// ---- POUs/PRG_IM1L1_PPM.TcPOU
PROGRAM PRG_IM1L1_PPM
VAR
    {attribute 'pytmc' := '
        pv: IM1L1:PPM
        io: io
    '}
    {attribute 'TcLinkTo' := '.fbGige.iIlluminatorINT := TIIB[IM1L1-EL4004]^AO Outputs Channel 1^Analog output;
                              .fbGige.bGigePower := TIIB[IM1L1-EL2004]^Channel 2^Output;
                              .fbPowerMeter.iVoltageINT := TIIB[IM1L1-EL3062]^AI Standard Channel 1^Value;
                              .fbPowerMeter.fbTempSensor.bError := TIIB[IM1L1-EL3314]^TC Inputs Channel 1^Status^Error;
                              .fbPowerMeter.fbTempSensor.bUnderrange := TIIB[IM1L1-EL3314]^TC Inputs Channel 1^Status^Underrange;
                              .fbPowerMeter.fbTempSensor.bOverrange := TIIB[IM1L1-EL3314]^TC Inputs Channel 1^Status^Overrange;
                              .fbPowerMeter.fbTempSensor.iRaw := TIIB[IM1L1-EL3314]^TC Inputs Channel 1^Value;
                              .fbYagTempSensor.bError := TIIB[IM1L1-EL3314]^TC Inputs Channel 2^Status^Error;
                              .fbYagTempSensor.bUnderrange := TIIB[IM1L1-EL3314]^TC Inputs Channel 2^Status^Underrange;
                              .fbYagTempSensor.bOverrange := TIIB[IM1L1-EL3314]^TC Inputs Channel 2^Status^Overrange;
                              .fbYagTempSensor.iRaw := TIIB[IM1L1-EL3314]^TC Inputs Channel 2^Value'}
    fbIM1L1: FB_PPM;

    fbStateSetup: FB_StateSetupHelper;
    stDefault: ST_PositionState := (
        fVelocity := 10,
        bMoveOk := TRUE,
        bValid := TRUE
    );
END_VAR


fbStateSetup(stPositionState:=stDefault, bSetDefault:=TRUE);
fbStateSetup(stPositionState:=fbIM1L1.stOut, fPosition:=-11,    sPmpsState:='IM1L1:PPM-OUT');
fbStateSetup(stPositionState:=fbIM1L1.stPower, fPosition:=-47.59, sPmpsState:='IM1L1:PPM-POWERMETER');
fbStateSetup(stPositionState:=fbIM1L1.stYag1, fPosition:=-71.69,  sPmpsState:='IM1L1:PPM-YAG1');
fbStateSetup(stPositionState:=fbIM1L1.stYag2, fPosition:=-97.70,  sPmpsState:='IM1L1:PPM-YAG2');

fbIM1L1(
    fbArbiter := GVL.fbArbiter2,
    fbFFHWO := GVL.fbFastFaultOutput2,
    stYStage := Main.M23,
    sDeviceName := 'IM1L1:PPM',
    sTransitionKey := 'IM1L1:PPM-TRANSITION',
    bEnableMotion := TRUE,
    bEnableBeamParams := TRUE,
    bEnablePositionLimits := TRUE,
    fResponsivity := 0.0640, //probably wrong, check with Phil
);

END_PROGRAM

// ---- POUs/PRG_IM2L0_XTES.TcPOU
PROGRAM PRG_IM2L0_XTES
VAR
    {attribute 'pytmc' := '
        pv: IM2L0:XTES
        io: io
    '}
    {attribute 'TcLinkTo' := '.bZoomEndFwd := TIIB[IM2L0-EL1088]^Channel 1^Input;
                              .bZoomEndBwd := TIIB[IM2L0-EL1088]^Channel 2^Input;
                              .bFocusEndFwd := TIIB[IM2L0-EL1088]^Channel 3^Input;
                              .bFocusEndBwd := TIIB[IM2L0-EL1088]^Channel 4^Input;
                              .fbOpal.bOpalPower := TIIB[IM2L0-EL2004]^Channel 2^Output;
                              .fbLED.bLedPower := TIIB[IM2L0-EL2004]^Channel 3^Output'}
    fbIM2L0: FB_XPIM;
    {attribute 'TcLinkTo' := '.Status := TIIB[IM2L0-EL6002]^COM TxPDO-Map Inputs Channel 1^Status;
                              .D[0] := TIIB[IM2L0-EL6002]^COM TxPDO-Map Inputs Channel 1^Data In 0;
                              .D[1] := TIIB[IM2L0-EL6002]^COM TxPDO-Map Inputs Channel 1^Data In 1;
                              .D[2] := TIIB[IM2L0-EL6002]^COM TxPDO-Map Inputs Channel 1^Data In 2;
                              .D[3] := TIIB[IM2L0-EL6002]^COM TxPDO-Map Inputs Channel 1^Data In 3;
                              .D[4] := TIIB[IM2L0-EL6002]^COM TxPDO-Map Inputs Channel 1^Data In 4;
                              .D[5] := TIIB[IM2L0-EL6002]^COM TxPDO-Map Inputs Channel 1^Data In 5;
                              .D[6] := TIIB[IM2L0-EL6002]^COM TxPDO-Map Inputs Channel 1^Data In 6;
                              .D[7] := TIIB[IM2L0-EL6002]^COM TxPDO-Map Inputs Channel 1^Data In 7;
                              .D[8] := TIIB[IM2L0-EL6002]^COM TxPDO-Map Inputs Channel 1^Data In 8;
                              .D[9] := TIIB[IM2L0-EL6002]^COM TxPDO-Map Inputs Channel 1^Data In 9;
                              .D[10] := TIIB[IM2L0-EL6002]^COM TxPDO-Map Inputs Channel 1^Data In 10;
                              .D[11] := TIIB[IM2L0-EL6002]^COM TxPDO-Map Inputs Channel 1^Data In 11;
                              .D[12] := TIIB[IM2L0-EL6002]^COM TxPDO-Map Inputs Channel 1^Data In 12;
                              .D[13] := TIIB[IM2L0-EL6002]^COM TxPDO-Map Inputs Channel 1^Data In 13;
                              .D[14] := TIIB[IM2L0-EL6002]^COM TxPDO-Map Inputs Channel 1^Data In 14;
                              .D[15] := TIIB[IM2L0-EL6002]^COM TxPDO-Map Inputs Channel 1^Data In 15;
                              .D[16] := TIIB[IM2L0-EL6002]^COM TxPDO-Map Inputs Channel 1^Data In 16;
                              .D[17] := TIIB[IM2L0-EL6002]^COM TxPDO-Map Inputs Channel 1^Data In 17;
                              .D[18] := TIIB[IM2L0-EL6002]^COM TxPDO-Map Inputs Channel 1^Data In 18;
                              .D[19] := TIIB[IM2L0-EL6002]^COM TxPDO-Map Inputs Channel 1^Data In 19;
                              .D[20] := TIIB[IM2L0-EL6002]^COM TxPDO-Map Inputs Channel 1^Data In 20;
                              .D[21] := TIIB[IM2L0-EL6002]^COM TxPDO-Map Inputs Channel 1^Data In 21'}
    stEL6In AT %I*: EL6InData22b;
    {attribute 'TcLinkTo' := '.Ctrl := TIIB[IM2L0-EL6002]^COM RxPDO-Map Outputs Channel 1^Ctrl;
                              .D[0] := TIIB[IM2L0-EL6002]^COM RxPDO-Map Outputs Channel 1^Data Out 0;
                              .D[1] := TIIB[IM2L0-EL6002]^COM RxPDO-Map Outputs Channel 1^Data Out 1;
                              .D[2] := TIIB[IM2L0-EL6002]^COM RxPDO-Map Outputs Channel 1^Data Out 2;
                              .D[3] := TIIB[IM2L0-EL6002]^COM RxPDO-Map Outputs Channel 1^Data Out 3;
                              .D[4] := TIIB[IM2L0-EL6002]^COM RxPDO-Map Outputs Channel 1^Data Out 4;
                              .D[5] := TIIB[IM2L0-EL6002]^COM RxPDO-Map Outputs Channel 1^Data Out 5;
                              .D[6] := TIIB[IM2L0-EL6002]^COM RxPDO-Map Outputs Channel 1^Data Out 6;
                              .D[7] := TIIB[IM2L0-EL6002]^COM RxPDO-Map Outputs Channel 1^Data Out 7;
                              .D[8] := TIIB[IM2L0-EL6002]^COM RxPDO-Map Outputs Channel 1^Data Out 8;
                              .D[9] := TIIB[IM2L0-EL6002]^COM RxPDO-Map Outputs Channel 1^Data Out 9;
                              .D[10] := TIIB[IM2L0-EL6002]^COM RxPDO-Map Outputs Channel 1^Data Out 10;
                              .D[11] := TIIB[IM2L0-EL6002]^COM RxPDO-Map Outputs Channel 1^Data Out 11;
                              .D[12] := TIIB[IM2L0-EL6002]^COM RxPDO-Map Outputs Channel 1^Data Out 12;
                              .D[13] := TIIB[IM2L0-EL6002]^COM RxPDO-Map Outputs Channel 1^Data Out 13;
                              .D[14] := TIIB[IM2L0-EL6002]^COM RxPDO-Map Outputs Channel 1^Data Out 14;
                              .D[15] := TIIB[IM2L0-EL6002]^COM RxPDO-Map Outputs Channel 1^Data Out 15;
                              .D[16] := TIIB[IM2L0-EL6002]^COM RxPDO-Map Outputs Channel 1^Data Out 16;
                              .D[17] := TIIB[IM2L0-EL6002]^COM RxPDO-Map Outputs Channel 1^Data Out 17;
                              .D[18] := TIIB[IM2L0-EL6002]^COM RxPDO-Map Outputs Channel 1^Data Out 18;
                              .D[19] := TIIB[IM2L0-EL6002]^COM RxPDO-Map Outputs Channel 1^Data Out 19;
                              .D[20] := TIIB[IM2L0-EL6002]^COM RxPDO-Map Outputs Channel 1^Data Out 20;
                              .D[21] := TIIB[IM2L0-EL6002]^COM RxPDO-Map Outputs Channel 1^Data Out 21'}
    stEL6Out AT %Q*: EL6OutData22b;

    fbStateSetup: FB_StateSetupHelper;
    stDefault: ST_PositionState := (
        fVelocity := 1,
        bMoveOk := TRUE,
        bValid := TRUE
    );

    {attribute 'TcLinkTo' := 'TIIB[IM2L0-EL7041]^STM Status^Status^Digital input 1'}
    bDefectiveLimitSwitch AT %I*: BOOL;
END_VAR


fbStateSetup(stPositionState:=stDefault, bSetDefault:=TRUE);
fbStateSetup(stPositionState:=fbIM2L0.stOut, fPosition:=0,          sPmpsState:='IM2L0:XTES-OUT');
fbStateSetup(stPositionState:=fbIM2L0.stYag, fPosition:=-87.65,     sPmpsState:='IM2L0:XTES-YAG');
fbStateSetup(stPositionState:=fbIM2L0.stDiamond, fPosition:=-57.65, sPmpsState:='IM2L0:XTES-DIAMOND');
fbStateSetup(stPositionState:=fbIM2L0.stReticle, fPosition:=-27.65, sPmpsState:='IM2L0:XTES-RETICLE');

Main.M24.bLimitForwardEnable := bDefectiveLimitSwitch OR (Main.M24.stAxisStatus.fActPosition < 0);

fbIM2L0(
    fbArbiter := GVL.fbArbiter,
    fbFFHWO := GVL.fbFastFaultOutput1,
    stYStage := Main.M24,
    stZoomStage := Main.M25,
    stFocusStage := Main.M26,
    stEl6In := stEL6In,
    stEl6Out := stEl6Out,
    sDeviceName := 'IM2L0:XTES',
    sTransitionKey := 'IM2L0:XTES-TRANSITION',
    bEnableMotion := TRUE,
    bEnableBeamParams := TRUE,
    bEnablePositionLimits := TRUE,
);

END_PROGRAM

// ---- POUs/PRG_IM3L0_PPM.TcPOU
PROGRAM PRG_IM3L0_PPM
VAR
    {attribute 'pytmc' := '
        pv: IM3L0:PPM
        io: io
    '}
    {attribute 'TcLinkTo' := '.fbGige.iIlluminatorINT := TIIB[IM3L0-EL4004]^AO Outputs Channel 1^Analog output;
                              .fbGige.bGigePower := TIIB[IM3L0-EL2004]^Channel 2^Output;
                              .fbPowerMeter.iVoltageINT := TIIB[IM3L0-EL3062]^AI Standard Channel 1^Value;
                              .fbPowerMeter.fbTempSensor.bError := TIIB[IM3L0-EL3314]^TC Inputs Channel 1^Status^Error;
                              .fbPowerMeter.fbTempSensor.bUnderrange := TIIB[IM3L0-EL3314]^TC Inputs Channel 1^Status^Underrange;
                              .fbPowerMeter.fbTempSensor.bOverrange := TIIB[IM3L0-EL3314]^TC Inputs Channel 1^Status^Overrange;
                              .fbPowerMeter.fbTempSensor.iRaw := TIIB[IM3L0-EL3314]^TC Inputs Channel 1^Value;
                              .fbYagTempSensor.bError := TIIB[IM3L0-EL3314]^TC Inputs Channel 2^Status^Error;
                              .fbYagTempSensor.bUnderrange := TIIB[IM3L0-EL3314]^TC Inputs Channel 2^Status^Underrange;
                              .fbYagTempSensor.bOverrange := TIIB[IM3L0-EL3314]^TC Inputs Channel 2^Status^Overrange;
                              .fbYagTempSensor.iRaw := TIIB[IM3L0-EL3314]^TC Inputs Channel 2^Value'}
    fbIM3L0: FB_PPM;

    fbStateSetup: FB_StateSetupHelper;
    stDefault: ST_PositionState := (
        fVelocity := 10,
        bMoveOk := TRUE,
        bValid := TRUE
    );
END_VAR


fbStateSetup(stPositionState:=stDefault, bSetDefault:=TRUE);
fbStateSetup(stPositionState:=fbIM3L0.stOut, fPosition:=-8.40,    sPmpsState:='IM3L0:PPM-OUT');
fbStateSetup(stPositionState:=fbIM3L0.stPower, fPosition:=-47.40, sPmpsState:='IM3L0:PPM-POWERMETER');
fbStateSetup(stPositionState:=fbIM3L0.stYag1, fPosition:=-71.50,  sPmpsState:='IM3L0:PPM-YAG1');
fbStateSetup(stPositionState:=fbIM3L0.stYag2, fPosition:=-97.51,  sPmpsState:='IM3L0:PPM-YAG2');

fbIM3L0(
    fbArbiter := GVL.fbArbiter,
    fbFFHWO := GVL.fbFastFaultOutput1,
    stYStage := Main.M27,
    sDeviceName := 'IM3L0:PPM',
    sTransitionKey := 'IM3L0:PPM-TRANSITION',
    bEnableMotion := TRUE,
    bEnableBeamParams := TRUE,
    bEnablePositionLimits := TRUE,
    fResponsivity := 0.0506,
);

END_PROGRAM

// ---- POUs/PRG_IM4L0_XTES.TcPOU
PROGRAM PRG_IM4L0_XTES
VAR
    {attribute 'pytmc' := '
        pv: IM4L0:XTES
        io: io
    '}
    {attribute 'TcLinkTo' := '.bZoomEndFwd := TIIB[IM4L0-EL1088]^Channel 1^Input;
                              .bZoomEndBwd := TIIB[IM4L0-EL1088]^Channel 2^Input;
                              .bFocusEndFwd := TIIB[IM4L0-EL1088]^Channel 3^Input;
                              .bFocusEndBwd := TIIB[IM4L0-EL1088]^Channel 4^Input;
                              .fbOpal.bOpalPower := TIIB[IM4L0-EL2004]^Channel 2^Output;
                              .fbLED.bLedPower := TIIB[IM4L0-EL2004]^Channel 3^Output'}
    fbIM4L0: FB_XPIM;
    {attribute 'TcLinkTo' := '.Status := TIIB[IM4L0-EL6002]^COM TxPDO-Map Inputs Channel 1^Status;
                              .D[0] := TIIB[IM4L0-EL6002]^COM TxPDO-Map Inputs Channel 1^Data In 0;
                              .D[1] := TIIB[IM4L0-EL6002]^COM TxPDO-Map Inputs Channel 1^Data In 1;
                              .D[2] := TIIB[IM4L0-EL6002]^COM TxPDO-Map Inputs Channel 1^Data In 2;
                              .D[3] := TIIB[IM4L0-EL6002]^COM TxPDO-Map Inputs Channel 1^Data In 3;
                              .D[4] := TIIB[IM4L0-EL6002]^COM TxPDO-Map Inputs Channel 1^Data In 4;
                              .D[5] := TIIB[IM4L0-EL6002]^COM TxPDO-Map Inputs Channel 1^Data In 5;
                              .D[6] := TIIB[IM4L0-EL6002]^COM TxPDO-Map Inputs Channel 1^Data In 6;
                              .D[7] := TIIB[IM4L0-EL6002]^COM TxPDO-Map Inputs Channel 1^Data In 7;
                              .D[8] := TIIB[IM4L0-EL6002]^COM TxPDO-Map Inputs Channel 1^Data In 8;
                              .D[9] := TIIB[IM4L0-EL6002]^COM TxPDO-Map Inputs Channel 1^Data In 9;
                              .D[10] := TIIB[IM4L0-EL6002]^COM TxPDO-Map Inputs Channel 1^Data In 10;
                              .D[11] := TIIB[IM4L0-EL6002]^COM TxPDO-Map Inputs Channel 1^Data In 11;
                              .D[12] := TIIB[IM4L0-EL6002]^COM TxPDO-Map Inputs Channel 1^Data In 12;
                              .D[13] := TIIB[IM4L0-EL6002]^COM TxPDO-Map Inputs Channel 1^Data In 13;
                              .D[14] := TIIB[IM4L0-EL6002]^COM TxPDO-Map Inputs Channel 1^Data In 14;
                              .D[15] := TIIB[IM4L0-EL6002]^COM TxPDO-Map Inputs Channel 1^Data In 15;
                              .D[16] := TIIB[IM4L0-EL6002]^COM TxPDO-Map Inputs Channel 1^Data In 16;
                              .D[17] := TIIB[IM4L0-EL6002]^COM TxPDO-Map Inputs Channel 1^Data In 17;
                              .D[18] := TIIB[IM4L0-EL6002]^COM TxPDO-Map Inputs Channel 1^Data In 18;
                              .D[19] := TIIB[IM4L0-EL6002]^COM TxPDO-Map Inputs Channel 1^Data In 19;
                              .D[20] := TIIB[IM4L0-EL6002]^COM TxPDO-Map Inputs Channel 1^Data In 20;
                              .D[21] := TIIB[IM4L0-EL6002]^COM TxPDO-Map Inputs Channel 1^Data In 21'}
    stEL6In AT %I*: EL6InData22b;
    {attribute 'TcLinkTo' := '.Ctrl := TIIB[IM4L0-EL6002]^COM RxPDO-Map Outputs Channel 1^Ctrl;
                              .D[0] := TIIB[IM4L0-EL6002]^COM RxPDO-Map Outputs Channel 1^Data Out 0;
                              .D[1] := TIIB[IM4L0-EL6002]^COM RxPDO-Map Outputs Channel 1^Data Out 1;
                              .D[2] := TIIB[IM4L0-EL6002]^COM RxPDO-Map Outputs Channel 1^Data Out 2;
                              .D[3] := TIIB[IM4L0-EL6002]^COM RxPDO-Map Outputs Channel 1^Data Out 3;
                              .D[4] := TIIB[IM4L0-EL6002]^COM RxPDO-Map Outputs Channel 1^Data Out 4;
                              .D[5] := TIIB[IM4L0-EL6002]^COM RxPDO-Map Outputs Channel 1^Data Out 5;
                              .D[6] := TIIB[IM4L0-EL6002]^COM RxPDO-Map Outputs Channel 1^Data Out 6;
                              .D[7] := TIIB[IM4L0-EL6002]^COM RxPDO-Map Outputs Channel 1^Data Out 7;
                              .D[8] := TIIB[IM4L0-EL6002]^COM RxPDO-Map Outputs Channel 1^Data Out 8;
                              .D[9] := TIIB[IM4L0-EL6002]^COM RxPDO-Map Outputs Channel 1^Data Out 9;
                              .D[10] := TIIB[IM4L0-EL6002]^COM RxPDO-Map Outputs Channel 1^Data Out 10;
                              .D[11] := TIIB[IM4L0-EL6002]^COM RxPDO-Map Outputs Channel 1^Data Out 11;
                              .D[12] := TIIB[IM4L0-EL6002]^COM RxPDO-Map Outputs Channel 1^Data Out 12;
                              .D[13] := TIIB[IM4L0-EL6002]^COM RxPDO-Map Outputs Channel 1^Data Out 13;
                              .D[14] := TIIB[IM4L0-EL6002]^COM RxPDO-Map Outputs Channel 1^Data Out 14;
                              .D[15] := TIIB[IM4L0-EL6002]^COM RxPDO-Map Outputs Channel 1^Data Out 15;
                              .D[16] := TIIB[IM4L0-EL6002]^COM RxPDO-Map Outputs Channel 1^Data Out 16;
                              .D[17] := TIIB[IM4L0-EL6002]^COM RxPDO-Map Outputs Channel 1^Data Out 17;
                              .D[18] := TIIB[IM4L0-EL6002]^COM RxPDO-Map Outputs Channel 1^Data Out 18;
                              .D[19] := TIIB[IM4L0-EL6002]^COM RxPDO-Map Outputs Channel 1^Data Out 19;
                              .D[20] := TIIB[IM4L0-EL6002]^COM RxPDO-Map Outputs Channel 1^Data Out 20;
                              .D[21] := TIIB[IM4L0-EL6002]^COM RxPDO-Map Outputs Channel 1^Data Out 21'}
    stEL6Out AT %Q*: EL6OutData22b;

     {attribute 'pytmc' := 'pv: IM4L0:SCRP:LED:01:PWR
                        io: io
                        field: ZNAM OFF
                        field: ONAM ON
     '}

     {attribute 'TcLinkTo' := 'TIIB[IM4L0-EL2004]^Channel 4^Output'}
    bIM4L0_SCRP_LED_01 AT %Q*: BOOL;

    fbStateSetup: FB_StateSetupHelper;
    stDefault: ST_PositionState := (
        fVelocity := 1,
        bMoveOk := TRUE,
        bValid := TRUE
    );
END_VAR


fbStateSetup(stPositionState:=stDefault, bSetDefault:=TRUE);
fbStateSetup(stPositionState:=fbIM4L0.stOut, fPosition:=0,          sPmpsState:='IM4L0:XTES-OUT');
fbStateSetup(stPositionState:=fbIM4L0.stYag, fPosition:=-86.65,     sPmpsState:='IM4L0:XTES-YAG');
fbStateSetup(stPositionState:=fbIM4L0.stDiamond, fPosition:=-56.65, sPmpsState:='IM4L0:XTES-DIAMOND');
fbStateSetup(stPositionState:=fbIM4L0.stReticle, fPosition:=-26.65, sPmpsState:='IM4L0:XTES-RETICLE');

fbIM4L0(
    fbArbiter := GVL.fbArbiter,
    fbFFHWO := GVL.fbFastFaultOutput1,
    stYStage := Main.M28,
    stZoomStage := Main.M29,
    stFocusStage := Main.M30,
    stEl6In := stEL6In,
    stEl6Out := stEl6Out,
    sDeviceName := 'IM4L0:XTES',
    sTransitionKey := 'IM4L0:XTES-TRANSITION',
    bEnableMotion := TRUE,
    bEnableBeamParams := TRUE,
    bEnablePositionLimits := TRUE,
);

END_PROGRAM

// ---- POUs/PRG_PF1L0_WFS.TcPOU
PROGRAM PRG_PF1L0_WFS
VAR
    {attribute 'pytmc' := '
        pv: PF1L0:WFS
        io: io
    '}
    {attribute 'TcLinkTo' := '.fbThermoCouple1.bError := TIIB[PF1L0-EL3314]^TC Inputs Channel 1^Status^Error;
                              .fbThermoCouple1.bUnderrange := TIIB[PF1L0-EL3314]^TC Inputs Channel 1^Status^Underrange;
                              .fbThermoCouple1.bOverrange := TIIB[PF1L0-EL3314]^TC Inputs Channel 1^Status^Overrange;
                              .fbThermoCouple1.iRaw := TIIB[PF1L0-EL3314]^TC Inputs Channel 1^Value;
                              .fbThermoCouple2.bError := TIIB[PF1L0-EL3314]^TC Inputs Channel 2^Status^Error;
                              .fbThermoCouple2.bUnderrange := TIIB[PF1L0-EL3314]^TC Inputs Channel 2^Status^Underrange;
                              .fbThermoCouple2.bOverrange := TIIB[PF1L0-EL3314]^TC Inputs Channel 2^Status^Overrange;
                              .fbThermoCouple2.iRaw := TIIB[PF1L0-EL3314]^TC Inputs Channel 2^Value'}
    fbPF1L0: FB_WFS;
    stSiBP: ST_BeamParams := PMPS_GVL.cstFullBeam;
    stFoilBP: ST_BeamParams := PMPS_GVL.cstFullBeam;

    fbStateSetup: FB_StateSetupHelper;
    stDefault: ST_PositionState := (
        fVelocity := 1,
        bMoveOk := TRUE,
        bValid := TRUE
    );
END_VAR


fbStateSetup(stPositionState:=stDefault, bSetDefault:=TRUE);
fbStateSetup(stPositionState:=fbPF1L0.stOut, fPosition:=-13,         sPmpsState:='PF1L0:WFS-OUT');
fbStateSetup(stPositionState:=fbPF1L0.stTarget1, fPosition:=-93.77,  sPmpsState:='PF1L0:WFS-TARGET1');
fbStateSetup(stPositionState:=fbPF1L0.stTarget2, fPosition:=-79.402, sPmpsState:='PF1L0:WFS-TARGET2');
fbStateSetup(stPositionState:=fbPF1L0.stTarget3, fPosition:=-65.028, sPmpsState:='PF1L0:WFS-TARGET3');
fbStateSetup(stPositionState:=fbPF1L0.stTarget4, fPosition:=-50.652, sPmpsState:='PF1L0:WFS-TARGET4');
fbStateSetup(stPositionState:=fbPF1L0.stTarget5, fPosition:=-36.277, sPmpsState:='PF1L0:WFS-TARGET5');

fbPF1L0(
    fbArbiter := GVL.fbArbiter,
    fbFFHWO := GVL.fbFastFaultOutput1,
    stYStage := Main.M31,
    stZStage := Main.M32,
    sDeviceName := 'PF1L0:WFS',
    sTransitionKey := 'PF1L0:WFS-TRANSITION',
    bEnableMotion := TRUE,
    bEnableBeamParams := TRUE,
    bEnablePositionLimits := TRUE,
    eEnumGet => GVL.ePF1L0State,
);

END_PROGRAM

// ---- POUs/PRG_RTDSL0.TcPOU
PROGRAM PRG_RTDSL0
VAR

    fbRTDSL0_Diode_MMS_01: FB_MotionStage;

    bInit: BOOL := TRUE;
END_VAR

// Placeholder, standard simulated motion for all axes
//fbMotion1(stMotionStage := Main.M33);
//fbMotion2(stMotionStage := Main.M34);
//fbMotion3(stMotionStage := Main.M35);
//fbMotion4(stMotionStage := Main.M36);
//fbMotion5(stMotionStage := Main.M37);
//fbMotion6(stMotionStage := Main.M38);
//fbMotion7(stMotionStage := Main.M39);

//Pneumatic actuators - OTR filters

RTDSL0_MPA_01(
    ibInsertOK:= TRUE,
    ibRetractOK:= TRUE ,
    ibPMPS_OK:= TRUE ,
    ibOverrideInterlock:= ,
    q_stAct=> ,
    xMPS_OK=> ,
    xDone=> ,
    i_xReset := ,
    io_fbFFHWO := GVL.fbFastFaultOutput1,
    bEnableFF := TRUE,
);

RTDSL0_MPA_02(
    ibInsertOK:= TRUE,
    ibRetractOK:= TRUE ,
    ibPMPS_OK:= TRUE ,
    ibOverrideInterlock:= ,
    q_stAct=> ,
    xMPS_OK=> ,
    xDone=> ,
    i_xReset := ,
    io_fbFFHWO := GVL.fbFastFaultOutput1,
    bEnableFF := TRUE,
);

RTDSL0_MPA_03(
    ibInsertOK:= TRUE,
    ibRetractOK:= TRUE ,
    ibPMPS_OK:= TRUE ,
    ibOverrideInterlock:= ,
    q_stAct=> ,
    xMPS_OK=> ,
    xDone=> ,
    i_xReset := ,
    io_fbFFHWO := GVL.fbFastFaultOutput1,
    bEnableFF := FALSE,
);
//  init the motion stages parameters
IF ( bInit) THEN
    Main.M33.bHardwareEnable := TRUE;
    Main.M33.bPowerSelf :=TRUE;
    Main.M33.nBrakeMode := ENUM_StageBrakeMode.NO_BRAKE;
    (* uncomment when mccallister goes from RTDSK0 -> RTDSL0
    Main.M34.bHardwareEnable := TRUE;
    Main.M34.bPowerSelf :=TRUE;
    Main.M34.nBrakeMode := ENUM_StageBrakeMode.NO_BRAKE;

    Main.M35.bHardwareEnable := TRUE;
    Main.M35.bPowerSelf :=TRUE;
    Main.M35.nBrakeMode := ENUM_StageBrakeMode.NO_BRAKE;

    Main.M36.bHardwareEnable := TRUE;
    Main.M36.bPowerSelf :=TRUE;
    Main.M36.nBrakeMode := ENUM_StageBrakeMode.NO_BRAKE;

    //LDM motor
    Main.M37.bHardwareEnable := TRUE;
    Main.M37.bPowerSelf :=TRUE;
    Main.M37.nBrakeMode := ENUM_StageBrakeMode.NO_BRAKE;
    *)
    Main.M33.nHomingMode := ENUM_EpicsHomeCmd.HIGH_LIMIT;
    //uncomment when mccallister gets moved RTDSK0->RTDSL0
    //Main.M34.nHomingMode := ENUM_EpicsHomeCmd.HIGH_LIMIT;
    //Main.M35.nHomingMode := ENUM_EpicsHomeCmd.HIGH_LIMIT;
    //Main.M36.nHomingMode := ENUM_EpicsHomeCmd.HIGH_LIMIT;
    Main.M37.nHomingMode := ENUM_EpicsHomeCmd.HIGH_LIMIT;

        bInit := FALSE;

END_IF


fbRTDSL0_Diode_MMS_01 (stMotionStage := Main.M33);
//uncomment when mccallister stage RTDSK0 -> RTDSL0
//fbRTDSL0_SCRP_MMS_01 (stMotionStage := Main.M34);
//fbRTDSL0_SCRP_MMS_02 (stMotionStage := Main.M35);
//fbRTDSL0_SCRP_MMS_03 (stMotionStage := Main.M36);
//fbRTDSL0_LDM_MMS_01 (stMotionStage := Main.M37);
//uncomment when mccallister stage RTDSK0->RTDSL0
//fbRTDSK0_SCRP_LED_01 (enumXPIM := Main.LED1);

END_PROGRAM

// ---- POUs/PRG_SL1L0_POWER.TcPOU
PROGRAM PRG_SL1L0_POWER
VAR // fix linking to rtd in the following order Bottom - South - TOP - NORTH
    {attribute 'pytmc' := '
        pv: SL1L0:POWER
        io: io
    '}
    {attribute 'TcLinkTo' := '.RTD_Bottom_1.iRaw := TIIB[SL1L0-EL3202-E8]^RTD Inputs Channel 1^Value;
                              .RTD_Bottom_1.bError := TIIB[SL1L0-EL3202-E8]^RTD Inputs Channel 1^Status^Error;
                              .RTD_Bottom_1.bUnderrange := TIIB[SL1L0-EL3202-E8]^RTD Inputs Channel 1^Status^Underrange;
                              .RTD_Bottom_1.bOverrange := TIIB[SL1L0-EL3202-E8]^RTD Inputs Channel 1^Status^Overrange;
                              .RTD_Bottom_2.iRaw := TIIB[SL1L0-EL3202-E8]^RTD Inputs Channel 2^Value;
                              .RTD_Bottom_2.bError := TIIB[SL1L0-EL3202-E8]^RTD Inputs Channel 2^Status^Error;
                              .RTD_Bottom_2.bUnderrange := TIIB[SL1L0-EL3202-E8]^RTD Inputs Channel 2^Status^Underrange;
                              .RTD_Bottom_2.bOverrange := TIIB[SL1L0-EL3202-E8]^RTD Inputs Channel 2^Status^Overrange;
                              .RTD_South_1.iRaw := TIIB[SL1L0-EL3202-E9]^RTD Inputs Channel 1^Value;
                              .RTD_South_1.bError := TIIB[SL1L0-EL3202-E9]^RTD Inputs Channel 1^Status^Error;
                              .RTD_South_1.bUnderrange := TIIB[SL1L0-EL3202-E9]^RTD Inputs Channel 1^Status^Underrange;
                              .RTD_South_1.bOverrange := TIIB[SL1L0-EL3202-E9]^RTD Inputs Channel 1^Status^Overrange;
                              .RTD_South_2.iRaw := TIIB[SL1L0-EL3202-E9]^RTD Inputs Channel 2^Value;
                              .RTD_South_2.bError := TIIB[SL1L0-EL3202-E9]^RTD Inputs Channel 2^Status^Error;
                              .RTD_South_2.bUnderrange := TIIB[SL1L0-EL3202-E9]^RTD Inputs Channel 2^Status^Underrange;
                              .RTD_South_2.bOverrange := TIIB[SL1L0-EL3202-E9]^RTD Inputs Channel 2^Status^Overrange;
                              .RTD_TOP_1.iRaw := TIIB[SL1L0-EL3202-E10]^RTD Inputs Channel 1^Value;
                              .RTD_TOP_1.bError := TIIB[SL1L0-EL3202-E10]^RTD Inputs Channel 1^Status^Error;
                              .RTD_TOP_1.bUnderrange := TIIB[SL1L0-EL3202-E10]^RTD Inputs Channel 1^Status^Underrange;
                              .RTD_TOP_1.bOverrange := TIIB[SL1L0-EL3202-E10]^RTD Inputs Channel 1^Status^Overrange;
                              .RTD_TOP_2.iRaw := TIIB[SL1L0-EL3202-E10]^RTD Inputs Channel 2^Value;
                              .RTD_TOP_2.bError := TIIB[SL1L0-EL3202-E10]^RTD Inputs Channel 2^Status^Error;
                              .RTD_TOP_2.bUnderrange := TIIB[SL1L0-EL3202-E10]^RTD Inputs Channel 2^Status^Underrange;
                              .RTD_TOP_2.bOverrange := TIIB[SL1L0-EL3202-E10]^RTD Inputs Channel 2^Status^Overrange;
                              .RTD_North_1.iRaw := TIIB[SL1L0-EL3202-E11]^RTD Inputs Channel 1^Value;
                              .RTD_North_1.bError := TIIB[SL1L0-EL3202-E11]^RTD Inputs Channel 1^Status^Error;
                              .RTD_North_1.bUnderrange := TIIB[SL1L0-EL3202-E11]^RTD Inputs Channel 1^Status^Underrange;
                              .RTD_North_1.bOverrange := TIIB[SL1L0-EL3202-E11]^RTD Inputs Channel 1^Status^Overrange;
                              .RTD_North_2.iRaw := TIIB[SL1L0-EL3202-E11]^RTD Inputs Channel 2^Value;
                              .RTD_North_2.bError := TIIB[SL1L0-EL3202-E11]^RTD Inputs Channel 2^Status^Error;
                              .RTD_North_2.bUnderrange := TIIB[SL1L0-EL3202-E11]^RTD Inputs Channel 2^Status^Underrange;
                              .RTD_North_2.bOverrange := TIIB[SL1L0-EL3202-E11]^RTD Inputs Channel 2^Status^Overrange'}
    fbSL1L0: FB_SLITS_POWER;

    {attribute 'pytmc' := '
    pv: SL1L0:POWER:GO;
    io: io;
    field: ZNAM False;
    field: ONAM True;
    '}
    bExecuteMotion:BOOL ;

    // Default True until it is properly linked to PMPS bit
    bMoveOk:BOOL :=TRUE;


    mcPower : ARRAY [1..4] OF MC_POWER;

        (*Offsets*)
    (* Absolute encoder value at the HLS + Absolute encoder value at the centered beam *)
    rEncoderOffsetTop: REAL := 15.55;
    rEncoderOffsetBottom: REAL := -12.99;
    rEncoderOffsetNorth: REAL := 12.2;
    rEncoderOffsetSouth: REAL := -16.8;

END_VAR



(*
--MAPPING TO PHYSICAL TERMINAL--
Main.41 -> M1    (Bottom)
Main.42 -> M2    (South)
Main.43 -> M3    (Top)
Main.44 -> M4    (North)
*)

fbSL1L0.rEncoderOffsetTop := rEncoderOffsetTop;
fbSL1L0.rEncoderOffsetBottom := rEncoderOffsetBottom;
fbSL1L0.rEncoderOffsetNorth := rEncoderOffsetNorth;
fbSL1L0.rEncoderOffsetSouth := rEncoderOffsetSouth;

//fbSL1L0.bExecuteMotion := bExecuteMotion;
fbSL1L0.bMoveOk := bMoveOk;
fbSL1L0(stTopBlade:=  Main.M43,
        stBottomBlade:= Main.M41,
        stNorthBlade:=  Main.M44,
        stSouthBlade:=  Main.M42,
        bExecuteMotion:=bExecuteMotion,
        io_fbFFHWO := GVL.fbFastFaultOutput1,
        fbArbiter := GVL.fbArbiter,
);
//fbSL1L0.M_UpdatePMPS(1); Not sure what index to use

//for testing purposes only. comment-out/delete once done.
(*mcPower[1](axis:=Main.M41.Axis, Enable:=TRUE, enable_positive:=Main.M41.bLimitForwardEnable, enable_negative:=Main.M41.bLimitBackwardEnable);
mcPower[2](axis:=Main.M42.Axis, Enable:=TRUE, enable_positive:=Main.M42.bLimitForwardEnable, enable_negative:=Main.M42.bLimitBackwardEnable);
mcPower[3](axis:=Main.M43.Axis, Enable:=TRUE, enable_positive:=Main.M43.bLimitForwardEnable, enable_negative:=Main.M43.bLimitBackwardEnable);
mcPower[4](axis:=Main.M44.Axis, Enable:=TRUE, enable_positive:=Main.M44.bLimitForwardEnable, enable_negative:=Main.M44.bLimitBackwardEnable);*)

END_PROGRAM

// ---- Temp/FB_SLITS_POWER.TcPOU
FUNCTION_BLOCK FB_SLITS_POWER EXTENDS FB_SLITS
VAR_INPUT
END_VAR
VAR
     {attribute 'pytmc' := '
        pv: FSW
    '}
    fbFlowSwitch: FB_XTES_Flowswitch;


    //RTDs
    {attribute 'pytmc' := '
        pv: TOP:RTD:01
    '}
    RTD_TOP_1: FB_TempSensor;
    {attribute 'pytmc' := '
        pv: TOP:RTD:02
    '}
    RTD_TOP_2: FB_TempSensor;
    {attribute 'pytmc' := '
        pv: BOTTOM:RTD:01
    '}
    RTD_Bottom_1: FB_TempSensor;
    {attribute 'pytmc' := '
        pv: BOTTOM:RTD:02
    '}
    RTD_Bottom_2: FB_TempSensor;

    {attribute 'pytmc' := '
        pv: NORTH:RTD:01
    '}
    RTD_North_1: FB_TempSensor;
    {attribute 'pytmc' := '
        pv: NORTH:RTD:02
    '}
    RTD_North_2: FB_TempSensor;
    {attribute 'pytmc' := '
        pv: SOUTH:RTD:01
    '}
    RTD_South_1: FB_TempSensor;
    {attribute 'pytmc' := '
        pv: SOUTH:RTD:02
    '}
    RTD_South_2: FB_TempSensor;


END_VAR

ACT_init();

// Instantiate Function block for all the blades
ACT_Motion();
//SET and GET the requested and Actual values
ACT_CalculatePositions();
//ACT_Zero();
//ACT_BLOCK();
ACT_RTDs();

ACTION ACT_RTDs:
////RTDs
RTD_TOP_1();
RTD_TOP_2();
RTD_Bottom_1();
RTD_Bottom_2();
RTD_North_1();
RTD_North_2();
RTD_South_1();
RTD_South_2();

//Flow Switch
fbFlowSwitch();
END_ACTION

END_FUNCTION_BLOCK

// ---- Temp/FB_SLITS.TcPOU
FUNCTION_BLOCK FB_SLITS
VAR_IN_OUT
    stTopBlade: DUT_MotionStage;
    stBottomBlade: DUT_MotionStage;
    stNorthBlade: DUT_MotionStage;
    stSouthBlade: DUT_MotionStage;
    bExecuteMotion:BOOL ;
END_VAR

VAR_INPUT

    {attribute 'pytmc' := '
    pv: PMPS_OK;
    io: i;
    field: ZNAM False
    field: ONAM True
    '}
    bMoveOk:BOOL;
    (*Offsets*)
    {attribute 'pytmc' := '
    pv: Offset_Top;
    io: io;
    '}
    rEncoderOffsetTop: REAL;
    {attribute 'pytmc' := '
    pv: ZeroOffset_Bottom;
    io: io;
    '}
    rEncoderOffsetBottom: REAL;
    {attribute 'pytmc' := '
    pv: ZeroOffset_North;
    io: io;
    '}
    rEncoderOffsetNorth: REAL;
    {attribute 'pytmc' := '
    pv: ZeroOffset_South;
    io: io;
    '}
    rEncoderOffsetSouth: REAL;
END_VAR

VAR
    fbTopBlade: FB_MotionStage;
    fbBottomBlade: FB_MotionStage;
    fbNorthBlade: FB_MotionStage;
    fbSouthBlade: FB_MotionStage;
    fPosTopBlade: LREAL;
    fPosBottomBlade: LREAL;
    fPosNorthBlade: LREAL;
    fPosSouthBlade: LREAL;

    (*Motion Parameters*)
    fSmallDelta: LREAL := 0.01;
    fBigDelta: LREAL := 10;
    fMaxVelocity: LREAL := 0.2;
    fHighAccel: LREAL := 0.8;
    fLowAccel: LREAL := 0.1;

    stTop: DUT_PositionState;
    stBOTTOM: DUT_PositionState;
    stNorth: DUT_PositionState;
    stSouth: DUT_PositionState;

    {attribute 'pytmc' := 'pv: TOP'}
    fbTop: FB_StatePTPMove;
    {attribute 'pytmc' := 'pv: BOTTOM'}
    fbBottom: FB_StatePTPMove;
    {attribute 'pytmc' := 'pv: NORTH'}
    fbNorth: FB_StatePTPMove;
    {attribute 'pytmc' := 'pv: SOUTH'}
    fbSouth: FB_StatePTPMove;

    (*EPICS pvs*)
    {attribute 'pytmc' := '
    pv: XWID_REQ;
    io: io;
    '}
    rReqApertureSizeX : REAL;
    {attribute 'pytmc' := '
    pv: YWID_REQ;
    io: io;
    '}
    rReqApertureSizeY : REAL;
    {attribute 'pytmc' := '
    pv: XCEN_REQ;
    io: io;
    '}
    rReqCenterX: REAL;
    {attribute 'pytmc' := '
    pv: YCEN_REQ;
    io: io;
    '}
    rReqCenterY: REAL;

    {attribute 'pytmc' := '
    pv: ACTUAL_XWIDTH;
    io: io;
    '}
    rActApertureSizeX : REAL;

    {attribute 'pytmc' := '
    pv: ACTUAL_YWIDTH;
    io: io;
    '}
    rActApertureSizeY : REAL;
    {attribute 'pytmc' := '
    pv: ACTUAL_XCENTER;
    io: io;
    '}
    rActCenterX: REAL;
    {attribute 'pytmc' := '
    pv: ACTUAL_YCENTER;
    io: io;
    '}
    rActCenterY: REAL;

    {attribute 'pytmc' := '
    pv: XCEN_SETZERO;
    io: io;
    '}
    rSetCenterX: BOOL;
    {attribute 'pytmc' := '
    pv: YCEN_SETZERO;
    io: io;
    '}
    rSetCenterY: BOOL;


    {attribute 'pytmc' := '
    pv: OPEN;
    io: io;
    field: ZNAM False
    field: ONAM True
    '}
    bOpen: BOOL;

    {attribute 'pytmc' := '
    pv: CLOSE;
    io: io;
    field: ZNAM False
    field: ONAM True
    '}
    bClose: BOOL;

    {attribute 'pytmc' := '
    pv: BLOCK;
    io: io;
    field: ZNAM False
    field: ONAM True
    '}
    bBlock: BOOL;



        //Local variables
    bInit: BOOL :=true;
    rTrig_Block: R_TRIG;
    rTrig_Open: R_TRIG;
    rTrig_Close: R_TRIG;

        //old values
    rOldReqApertureSizeX : REAL;
    rOldReqApertureSizeY : REAL;
    rOldReqCenterX: REAL;
    rOldReqCenterY: REAL;

    bExecuteMotionX: BOOL;
    bExecuteMotionY: BOOL;


    fPosBlock: LREAL;
    fPosClose: LREAL;
    fPosOpen: LREAL;

    stSetPositionOptions:ST_SetPositionOptions;
    fbSetPosition_TOP: MC_SetPosition;
    fbSetPosition_Bottom: MC_SetPosition;
    fbSetPosition_North: MC_SetPosition;
    fbSetPosition_South: MC_SetPosition;

    // For logging
    fbLogger : FB_LogMessage := (eSubsystem:=E_SubSystem.MOTION);

END_VAR

ACTION ACT_BLOCK:
rTrig_Block (CLK:= bBlock);
rTrig_Open (CLK:= bOpen);
rTrig_Close (CLK:= bClose);

if (rTrig_Block.Q) THEN
    //BLOCK

    bBlock := false;
END_IF

if (rTrig_Open.Q) THEN


    bOpen := false;
END_IF

if (rTrig_Close.Q) THEN


    bClose := false;
END_IF
END_ACTION

ACTION ACT_CalculatePositions:
//check if requested center or gap has changed
//check that the requested values are within acceptable motion range
IF (rOldReqApertureSizeX <> rReqApertureSizeX) THEN
    rOldReqApertureSizeX := rReqApertureSizeX;
    bExecuteMotionX := TRUE;
    fbLogger(sMsg:='Requested new X gap.', eSevr:=TcEventSeverity.Verbose);
END_IF

IF (rOldReqCenterX <> rReqCenterX) THEN
    rOldReqCenterX := rReqCenterX;
    bExecuteMotionX := TRUE;
    fbLogger(sMsg:='Requested new X center', eSevr:=TcEventSeverity.Verbose);

END_IF

IF (rOldReqApertureSizeY <> rReqApertureSizeY) THEN
    rOldReqApertureSizeY := rReqApertureSizeY;
    bExecuteMotionY := TRUE;
    fbLogger(sMsg:='Requested new Y gap.', eSevr:=TcEventSeverity.Verbose);
END_IF

IF (rOldReqCenterY <> rReqCenterY) THEN
   rOldReqCenterY := rReqCenterY;
   bExecuteMotionY := TRUE;
   fbLogger(sMsg:='Requested new Y center.', eSevr:=TcEventSeverity.Verbose);

END_IF


//Calculate requested target positions from requested gap and center
fPosTopBlade := (rReqApertureSizeY/2) + (rReqCenterY + rEncoderOffsetTop) ;
fPosBottomBlade := (-1*rReqApertureSizeY/2) + (rReqCenterY+rEncoderOffsetBottom);

fPosNorthBlade := (rReqApertureSizeX/2) + (rReqCenterX + rEncoderOffsetNorth);
fPosSouthBlade := (-1*rReqApertureSizeX/2) + (rReqCenterX + rEncoderOffsetSouth);


//Calculate actual gap and center from actual stages positions
rActApertureSizeX := LREAL_TO_REAL((stNorthBlade.stAxisStatus.fActPosition - rEncoderOffsetNorth) - (stSouthBlade.stAxisStatus.fActPosition- rEncoderOffsetSouth));

rActApertureSizeY := LREAL_TO_REAL((stTopBlade.stAxisStatus.fActPosition - rEncoderOffsetTop) - (stBottomBlade.stAxisStatus.fActPosition - rEncoderOffsetBottom));

rActCenterX := LREAL_TO_REAL((((stNorthBlade.stAxisStatus.fActPosition - rEncoderOffsetNorth)  + (stSouthBlade.stAxisStatus.fActPosition - rEncoderOffsetSouth ))/2));

rActCenterY := LREAL_TO_REAL((((stTopBlade.stAxisStatus.fActPosition - rEncoderOffsetTop) + (stBottomBlade.stAxisStatus.fActPosition - rEncoderOffsetBottom))/2));



//Update PMPS Arbiter with the Actual Size and Center of the Aperture
END_ACTION

ACTION ACT_Home:

END_ACTION

ACTION ACT_Init:

//  init the motion stages parameters
IF ( bInit) THEN
    stTopBlade.bHardwareEnable := TRUE;
    stBottomBlade.bHardwareEnable := TRUE;
    stNorthBlade.bHardwareEnable := TRUE;
    stSouthBlade.bHardwareEnable := TRUE;
    stTopBlade.bPowerSelf :=TRUE;
    stBottomBlade.bPowerSelf :=TRUE;
    stNorthBlade.bPowerSelf :=TRUE;
    stSouthBlade.bPowerSelf :=TRUE;
    stTopBlade.nBrakeMode := ENUM_StageBrakeMode.NO_BRAKE;
    stBottomBlade.nBrakeMode := ENUM_StageBrakeMode.NO_BRAKE;
    stNorthBlade.nBrakeMode := ENUM_StageBrakeMode.NO_BRAKE;
    stSouthBlade.nBrakeMode := ENUM_StageBrakeMode.NO_BRAKE;
END_IF
END_ACTION

ACTION ACT_Motion:
// Instantiate Function block for all the blades
fbTopBlade(stMotionStage:=stTopBlade);
fbBottomBlade(stMotionStage:=stBottomBlade);
fbNorthBlade(stMotionStage:=stNorthBlade);
fbSouthBlade(stMotionStage:=stSouthBlade);

// PTP Motion for each blade
stTop.sName := 'Top';
stTop.fPosition := fPosTopBlade;
stTop.fDelta := fSmallDelta;
stTop.fVelocity := fMaxVelocity;
stTop.fAccel := fHighAccel;
stTop.fDecel := fHighAccel;

stBOTTOM.sName := 'Bottom';
stBOTTOM.fPosition := fPosBottomBlade;
stBOTTOM.fDelta := fSmallDelta;
stBOTTOM.fVelocity := fMaxVelocity;
stBOTTOM.fAccel := fHighAccel;
stBOTTOM.fDecel := fHighAccel;

stNorth.sName := 'North';
stNorth.fPosition := fPosNorthBlade;
stNorth.fDelta := fSmallDelta;
stNorth.fVelocity := fMaxVelocity;
stNorth.fAccel := fHighAccel;
stNorth.fDecel := fHighAccel;

stSouth.sName := 'South';
stSouth.fPosition := fPosSouthBlade;
stSouth.fDelta := fSmallDelta;
stSouth.fVelocity := fMaxVelocity;
stSouth.fAccel := fHighAccel;
stSouth.fDecel := fHighAccel;

IF (bExecuteMotionY) THEN
    fbTop.bExecute := fbBottom.bExecute := bExecuteMotionY;
    bExecuteMotionY:= FALSE;
END_IF

IF (bExecuteMotionX) THEN
    fbNorth.bExecute := fbSouth.bExecute := bExecuteMotionX;
    bExecuteMotionX:= FALSE;
END_IF


fbTop(
    stPositionState:=stTop,
    bMoveOk:=bMoveOk,
    stMotionStage:=stTopBlade);

fbBottom(
    stPositionState:=stBOTTOM,
    bMoveOk:=bMoveOk,
    stMotionStage:=stBottomBlade);

fbNorth(
    stPositionState:=stNorth,
    bMoveOk:=bMoveOk,
    stMotionStage:=stNorthBlade);

fbSouth(
    stPositionState:=stSouth,
    bMoveOk:=bMoveOk,
    stMotionStage:=stSouthBlade);
END_ACTION

ACTION ACT_Zero:
//ZERO BIAS

// Set Y center to zero

// Set X center to zero

if (rSetCenterY)THEN
        rSetCenterY := false;
        // Set Current Position
        fbSetPosition_TOP.Position :=  stTopBlade.stAxisStatus.fActPosition - rActCenterY ;
        fbSetPosition_TOP.Execute := TRUE;
        fbSetPosition_Bottom.Position := stBottomBlade.stAxisStatus.fActPosition - rActCenterY;
        fbSetPosition_Bottom.Execute := TRUE;
END_IF

if (rSetCenterX)THEN
        rSetCenterX := false;
        // Set Current Position
        fbSetPosition_North.Position := stNorthBlade.stAxisStatus.fActPosition - rActCenterX ;
        fbSetPosition_North.Execute := TRUE;
        fbSetPosition_South.Position := stSouthBlade.stAxisStatus.fActPosition - rActCenterX ; ;
        fbSetPosition_South.Execute := TRUE;
END_IF


//Reset
if (fbSetPosition_TOP.Done ) THEN
    fbSetPosition_TOP.Execute := FALSE;
END_IF
if (fbSetPosition_Bottom.Done ) THEN
    fbSetPosition_Bottom.Execute := FALSE;
END_IF
if (fbSetPosition_North.Done ) THEN
    fbSetPosition_North.Execute := FALSE;
END_IF
if (fbSetPosition_South.Done ) THEN
    fbSetPosition_South.Execute := FALSE;
END_IF

// Set Encoder Position
//Clear position lag error
stSetPositionOptions.ClearPositionLag := TRUE;
fbSetPosition_TOP(
    Axis:=  stTopBlade.Axis ,
    Execute:= ,
    Position:= 0 ,
    Mode:= FALSE,
    Options:= stSetPositionOptions,
    Done=> ,
    Busy=> ,
    Error=> ,
    ErrorID=> );
fbSetPosition_Bottom(
    Axis:= stBottomBlade.Axis ,
    Execute:= ,
    Position:= 0 ,
    Mode:= FALSE,
    Options:= stSetPositionOptions,
    Done=> ,
    Busy=> ,
    Error=> ,
    ErrorID=> );
fbSetPosition_North(
    Axis:= stNorthBlade.Axis ,
    Execute:= ,
    Position:= 0 ,
    Mode:= FALSE,
    Options:= stSetPositionOptions,
    Done=> ,
    Busy=> ,
    Error=> ,
    ErrorID=> );
fbSetPosition_South(
    Axis:= stSouthBlade.Axis ,
    Execute:= ,
    Position:= 0 ,
    Mode:= FALSE,
    Options:= stSetPositionOptions,
    Done=> ,
    Busy=> ,
    Error=> ,
    ErrorID=> );
END_ACTION

END_FUNCTION_BLOCK

// ---- POUs/PRG_SL2L0_POWER.TcPOU
PROGRAM PRG_SL2L0_POWER
VAR // linking to rtd in the following order Bottom - South - TOP - NORTH
    {attribute 'pytmc' := '
        pv: SL2L0:POWER
        io: io
    '}
    {attribute 'TcLinkTo' := '.RTD_Bottom_1.iRaw := TIIB[SL2L0-EL3202-E8]^RTD Inputs Channel 1^Value;
                              .RTD_Bottom_1.bError := TIIB[SL2L0-EL3202-E8]^RTD Inputs Channel 1^Status^Error;
                              .RTD_Bottom_1.bUnderrange := TIIB[SL2L0-EL3202-E8]^RTD Inputs Channel 1^Status^Underrange;
                              .RTD_Bottom_1.bOverrange := TIIB[SL2L0-EL3202-E8]^RTD Inputs Channel 1^Status^Overrange;
                              .RTD_Bottom_2.iRaw := TIIB[SL2L0-EL3202-E8]^RTD Inputs Channel 2^Value;
                              .RTD_Bottom_2.bError := TIIB[SL2L0-EL3202-E8]^RTD Inputs Channel 2^Status^Error;
                              .RTD_Bottom_2.bUnderrange := TIIB[SL2L0-EL3202-E8]^RTD Inputs Channel 2^Status^Underrange;
                              .RTD_Bottom_2.bOverrange := TIIB[SL2L0-EL3202-E8]^RTD Inputs Channel 2^Status^Overrange;
                              .RTD_South_1.iRaw := TIIB[SL2L0-EL3202-E9]^RTD Inputs Channel 1^Value;
                              .RTD_South_1.bError := TIIB[SL2L0-EL3202-E9]^RTD Inputs Channel 1^Status^Error;
                              .RTD_South_1.bUnderrange := TIIB[SL2L0-EL3202-E9]^RTD Inputs Channel 1^Status^Underrange;
                              .RTD_South_1.bOverrange := TIIB[SL2L0-EL3202-E9]^RTD Inputs Channel 1^Status^Overrange;
                              .RTD_South_2.iRaw := TIIB[SL2L0-EL3202-E9]^RTD Inputs Channel 2^Value;
                              .RTD_South_2.bError := TIIB[SL2L0-EL3202-E9]^RTD Inputs Channel 2^Status^Error;
                              .RTD_South_2.bUnderrange := TIIB[SL2L0-EL3202-E9]^RTD Inputs Channel 2^Status^Underrange;
                              .RTD_South_2.bOverrange := TIIB[SL2L0-EL3202-E9]^RTD Inputs Channel 2^Status^Overrange;
                              .RTD_TOP_1.iRaw := TIIB[SL2L0-EL3202-E10]^RTD Inputs Channel 1^Value;
                              .RTD_TOP_1.bError := TIIB[SL2L0-EL3202-E10]^RTD Inputs Channel 1^Status^Error;
                              .RTD_TOP_1.bUnderrange := TIIB[SL2L0-EL3202-E10]^RTD Inputs Channel 1^Status^Underrange;
                              .RTD_TOP_1.bOverrange := TIIB[SL2L0-EL3202-E10]^RTD Inputs Channel 1^Status^Overrange;
                              .RTD_TOP_2.iRaw := TIIB[SL2L0-EL3202-E10]^RTD Inputs Channel 2^Value;
                              .RTD_TOP_2.bError := TIIB[SL2L0-EL3202-E10]^RTD Inputs Channel 2^Status^Error;
                              .RTD_TOP_2.bUnderrange := TIIB[SL2L0-EL3202-E10]^RTD Inputs Channel 2^Status^Underrange;
                              .RTD_TOP_2.bOverrange := TIIB[SL2L0-EL3202-E10]^RTD Inputs Channel 2^Status^Overrange;
                              .RTD_North_1.iRaw := TIIB[SL2L0-EL3202-E10]^RTD Inputs Channel 1^Value;
                              .RTD_North_1.bError := TIIB[SL2L0-EL3202-E10]^RTD Inputs Channel 1^Status^Error;
                              .RTD_North_1.bUnderrange := TIIB[SL2L0-EL3202-E11]^RTD Inputs Channel 1^Status^Underrange;
                              .RTD_North_1.bOverrange := TIIB[SL2L0-EL3202-E11]^RTD Inputs Channel 1^Status^Overrange;
                              .RTD_North_2.iRaw := TIIB[SL2L0-EL3202-E11]^RTD Inputs Channel 2^Value;
                              .RTD_North_2.bError := TIIB[SL2L0-EL3202-E11]^RTD Inputs Channel 2^Status^Error;
                              .RTD_North_2.bUnderrange := TIIB[SL2L0-EL3202-E11]^RTD Inputs Channel 2^Status^Underrange;
                              .RTD_North_2.bOverrange := TIIB[SL2L0-EL3202-E11]^RTD Inputs Channel 2^Status^Overrange'}
    fbSL2L0: FB_SLITS_POWER;

    {attribute 'pytmc' := '
    pv: SL2L0:POWER:GO;
    io: io;
    field: ZNAM False;
    field: ONAM True;
    '}
    bExecuteMotion:BOOL ;


    (*fbMotion1: FB_SimMotor;
    fbMotion2: FB_SimMotor;
    fbMotion3: FB_SimMotor;
    fbMotion4: FB_SimMotor;*)
    bMoveOk:BOOL :=TRUE;

     (*Offsets*)
    (* Absolute encoder value at the HLS + Absolute encoder value at the centered beam *)
    rEncoderOffsetTop: REAL := 0;
    rEncoderOffsetBottom: REAL := 0;
    rEncoderOffsetNorth: REAL := 0;
    rEncoderOffsetSouth: REAL := 0;

    fbSL1L0: INT;
END_VAR


(*
--MAPPING TO PHYSICAL TERMINAL--
Main.M45 -> M1    (Bottom)
Main.M46 -> M2    (South)
Main.M47 -> M3    (Top)
Main.M48 -> M4    (North)
*)

fbSL2L0.rEncoderOffsetTop := rEncoderOffsetTop;
fbSL2L0.rEncoderOffsetBottom := rEncoderOffsetBottom;
fbSL2L0.rEncoderOffsetNorth := rEncoderOffsetNorth;
fbSL2L0.rEncoderOffsetSouth := rEncoderOffsetSouth;

fbSL2L0.bMoveOk := bMoveOk;
fbSL2L0(stTopBlade:=  Main.M47,
        stBottomBlade:= Main.M45,
        stNorthBlade:=  Main.M48,
        stSouthBlade:=  Main.M46,
        bExecuteMotion:=bExecuteMotion,
        io_fbFFHWO := GVL.fbFastFaultOutput1,
        fbArbiter := GVL.fbArbiter,
);
//fbSL2L0.M_UpdatePMPS(1); Not sure what index to use

END_PROGRAM

// ---- POUs/PRG_3_PMPS_POST.TcPOU
PROGRAM PRG_3_PMPS_POST
VAR
    fbArbiterIO: FB_SubSysToArbiter_IO;
    bMR1L1_Veto_OUT: BOOL;
    fbVetoArbiter_L1: FB_VetoArbiter;
END_VAR

bMR1L1_Veto_OUT := PMPS_GVL.stCurrentBeamParameters.aVetoDevices[PMPS.L_Stopper.MR1L1_OUT] AND NOT PMPS_GVL.stCurrentBeamParameters.aVetoDevices[PMPS.L_Stopper.MR1L1_IN];

GVL.fbFastFaultOutput1.Execute();
GVL.fbFastFaultOutput2.Execute(i_xVeto:=bMR1L1_Veto_OUT);

fbVetoArbiter_L1(bVeto:=bMR1L1_Veto_OUT,
                HigherAuthority := GVL.fbArbiter,
                LowerAuthority := GVL.fbArbiter2,
                FFO := GVL.fbFastFaultOutput1);

fbArbiterIO(
    Arbiter:=GVL.fbArbiter,
    fbFFHWO:=GVL.fbFastFaultOutput1);

END_PROGRAM

// ---- POUs/PRG_4_LOG.TcPOU
PROGRAM PRG_4_LOG
VAR
    fbLogHandler: FB_LogHandler;
END_VAR

fbLogHandler();

END_PROGRAM

// ---- Temp/FB_MPA.TcPOU
FUNCTION_BLOCK FB_MPA
VAR_INPUT
    (*EPS Interlock Bits*)
    ibInsertOK: BOOL;
    ibRetractOK: BOOL;
    ibPMPS_OK:BOOL;
    ibOverrideInterlock:BOOL; (*if true interlocks are ignored*)
    // Reset fault
    {attribute 'pytmc' := '
    pv: FF_Reset
    '}
    i_xReset: BOOL;
    sName: STRING;
    bEnableFF: BOOL := TRUE;
END_VAR
VAR_OUTPUT
    {attribute 'pytmc' := '
    pv:
    '}
    q_stAct     :    ST_MPA;
    {attribute 'pytmc' := '
    pv: MPS_FAULT
    '}
    xMPS_OK:BOOL;
    {attribute 'pytmc' := '
    pv: MOT_DONE
    '}
    xDone:Bool; // Motion is Done
END_VAR
VAR_IN_OUT
    io_fbFFHWO    :    FB_HardwareFFOutput;
END_VAR
VAR
    // PMPS
    fbFF    :    FB_FastFault :=(
        i_xAutoReset := TRUE,
        i_Desc := 'Device is moving',
        i_TypeCode := 16#1010);

    (*Init*)
    xFirstPass    :    BOOL;
    fbFSInit        :    R_TRIG;

    (* Timeouts*)
    tTimeOutDuration: TIME:= T#5S;
    tInserttimeout: TON;
    tRetracttimeout:TON;

    (*IO*)
    i_xInsertedLS    AT%I*: BOOL;
    i_xRetractedLS    AT%I*: BOOL;
    q_xInsert_DO    AT%Q*: BOOL;
    q_xRetract_DO    AT%Q*: BOOL;

    (* Reset Triggers *)
    rtInsert: R_TRIG;
    rtRemove: R_TRIG;
END_VAR


(*Initialize*)
fbFSInit( CLK := TRUE, Q => xFirstPass);
(*IO Mapping*)
ACT_IO();

IF xFirstPass THEN
    q_stAct.eState := INVALID;
    q_stAct.bRetract_SW := FALSE;
    q_stAct.bInsert_SW := FALSE;
END_IF


(* Manage States*)
IF q_stAct.i_bInLS AND  q_stAct.i_bOutLS THEN
    q_stAct.eState:=INVALID;
ELSIF NOT q_stAct.i_bInLS AND q_stAct.i_bOutLS THEN
    q_stAct.eState:=RETRACTED;
ELSIF q_stAct.i_bInLS AND NOT q_stAct.i_bOutLS THEN
    q_stAct.eState:=INSERTED;
ELSIF NOT q_stAct.i_bInLS AND NOT q_stAct.i_bOutLS THEN
    q_stAct.eState:=MOVING;
ELSE
    q_stAct.eState:=INVALID;
END_IF

(*Set the Done signal*)
xDone := (q_stAct.bRetract_SW AND q_stAct.eState=RETRACTED) OR (q_stAct.eState=INSERTED AND q_stAct.bInsert_SW);


(*MPS FAULT*)
(**)
xMPS_OK := (q_stAct.bRetract_SW AND i_xRetractedLS) XOR (i_xInsertedLS AND q_stAct.bInsert_SW);
//xMPS_OK := i_xRetractedLS XOR i_xInsertedLS;
//xMPS_OK := (q_stAct.eState=RETRACTED) OR (q_stAct.eState=INSERTED);
//xMPS_OK := (q_stAct.eState=RETRACTED) ;

(*PMPS PERMISSION*)

(* Reset the other command bit when one goes high *)
rtInsert(CLK:=q_stAct.bInsert_SW);
IF rtInsert.Q THEN
    q_stAct.bRetract_SW := FALSE;
END_IF
rtRemove(CLK:=q_stAct.bRetract_SW);
IF rtRemove.Q THEN
    q_stAct.bInsert_SW := FALSE;
END_IF

(* Can't have bRetract_SW and  bInsert_SW both be true*)
If (q_stAct.bRetract_SW) and (q_stAct.bInsert_SW) THEN
    q_stAct.bRetract_SW := FALSE;
    q_stAct.bInsert_SW := FALSE;
END_IF

(* Make the state consistent if we can *)
IF NOT (q_stAct.bRetract_SW OR q_stAct.bInsert_SW) THEN
    IF q_stAct.eState = RETRACTED THEN
        q_stAct.bRetract_SW := TRUE;
    ELSIF q_stAct.eState = INSERTED THEN
        q_stAct.bInsert_SW := TRUE;
    END_IF
END_IF

q_stAct.bRetractOK := ibRetractOK;
q_stAct.bInsertOK := ibInsertOK;

(*Actuate the device*)
q_stAct.q_bRetract := q_stAct.bRetractOK AND q_stAct.bRetract_SW;
q_stAct.q_bInsert := q_stAct.bInsertOK AND q_stAct.bInsert_SW;

IF q_stAct.q_bInsert THEN
    q_stAct.q_bRetract := FALSE;
    q_stAct.bRetract_SW:= FALSE;
ELSIF q_stAct.q_bRetract THEN
    q_stAct.q_bInsert := FALSE;
    q_stAct.bInsert_SW:= FALSE;
END_IF;




(*Timers*)
tInserttimeout(IN:= q_stAct.q_bInsert, PT := tTimeOutDuration );
tRetracttimeout(IN:= q_stAct.q_bRetract, PT := tTimeOutDuration);

///Check moving postion timout
IF NOT q_stAct.i_bInLS AND tInserttimeout.Q THEN
    q_stAct.bErrorPresent := TRUE;
ELSIF NOT q_stAct.i_bOutLS AND tRetracttimeout.Q THEN
    q_stAct.bErrorPresent := TRUE;
END_IF

(*FAST FAULT*)
IF bEnableFF THEN
    fbFF(i_DevName := sName,
        i_xOK := xMPS_OK,
        i_xReset := i_xReset,
        io_fbFFHWO := io_fbFFHWO);
END_IF

(*Soft IO Mapping*)
ACT_IO();

ACTION ACT_IO:
(*Inputs*)
q_stAct.i_bInLS :=  i_xInsertedLS;
q_stAct.i_bOutLS := i_xRetractedLS;

(*outputs*)
q_xInsert_DO:=q_stAct.q_bInsert;
q_xRetract_DO:=q_stAct.q_bRetract;
END_ACTION

END_FUNCTION_BLOCK

// ---- POUs/PRG_SP1L0_KMONO.TcPOU
PROGRAM PRG_SP1L0_KMONO
VAR
    fbMotion1: FB_MotionStage;
    fbMotion2: FB_MotionStage;
    fbMotion3: FB_MotionStage;
    fbMotion4: FB_MotionStage;
    fbMotion5: FB_MotionStage;
    fbMotion6: FB_MotionStage;

    (*
    fbFFO2: FB_BasicMotionStageAltFFO := (sName := 'SP1L0:KMONO:MMS:02');
    fbFFO4: FB_BasicMotionStageFFO := (sName := 'SP1L0:KMONO:MMS:04');
    fbFFO6: FB_BasicMotionStageFFO := (sName := 'SP1L0:KMONO:MMS:06');
    *)
    stOkBeam: ST_BeamParams := PMPS_GVL.cstFullBeam;
    bEnergyOk: BOOL;

    fbXTALFFO: FB_FastFault;
    bXtalOut: BOOL;
    bXtalIn: BOOL;

    fbRetFFO: FB_FastFault;
    bRetOut: BOOL;

    fbDiodeFFOAtPos: FB_FastFault;
    fbDiodeFFOEnergy: FB_FastFault;
    bDiodeOut: BOOL;
    bDiodeIn: BOOL;

    bInit: BOOL := TRUE;
END_VAR


IF bInit THEN
    // Only allow 7.7-8.9 keV
    stOkBeam.neVRange := F_eVIncludeRange(7700, 8900);
    bInit := FALSE;
END_IF
bEnergyOK := F_SafeBPCompare(PMPS_GVL.stCurrentBeamParameters, stOkBeam);

// Motor 1 XTAL ANGLE X (SP1L0-KMONO-MMS-01)
Main.M49.bLimitForwardEnable  := TRUE;    //TRUE
Main.M49.bLimitBackwardEnable := TRUE;    //TRUE
Main.M49.nEnableMode          := Enum_StageEnableMode.ALWAYS;
Main.M49.bHardwareEnable      := TRUE;
Main.M49.bPowerSelf           := TRUE;
fbMotion1(stMotionStage:=Main.M49);

// Motor 2 XTAL VERT Y (SP1L0-KMONO-MMS-02)
//Main.M50.bLimitForwardEnable  := bM2CCWLimit;    //(+Y)
//Main.M50.bLimitBackwardEnable := bM2CWLimit;    //(-Y)
Main.M50.nEnableMode          := Enum_StageEnableMode.ALWAYS;
Main.M50.bHardwareEnable      := TRUE;
Main.M50.bPowerSelf           := TRUE;
fbMotion2(stMotionStage:=Main.M50);
//fbFFO2(stMotionStage := Main.M50,
//       fbFFHWO := GVL.fbFastFaultOutput1,
//       bFFOk := Main.M50.stAxisStatus.fActPosition < 0.1);
// Andy says trip if IN and not between 7.7 and 8.9 keV
// Andy says reset if IN and between 7.7 and 8.9 keV OR at OUT
// IN is >50, out is at 0 (+-2)
bXtalOut := Main.M50.stAxisStatus.fActPosition < 2;
bXtalIn := Main.M50.stAxisStatus.fActPosition > 50;

fbXTALFFO(
    i_xOK := bEnergyOk OR NOT bXtalIn,
    i_xReset := bXtalOut OR (bXtalIn AND bEnergyOk),
    i_xAutoReset := TRUE,
    i_DevName := Main.M50.sName,
    i_Desc := 'Unsafe eV Range: needs 7.7-8.9keV',
    io_fbFFHWO := GVL.fbFastFaultOutput1);

// Motor 3 RETICLE HORIZ X (SP1L0-KMONO-MMS-03)
//Main.M51.bLimitForwardEnable  := bM3CCWLimit;    //(+X)
//Main.M51.bLimitBackwardEnable := bM3CWLimit;    //(-X)
Main.M51.nEnableMode          := Enum_StageEnableMode.DURING_MOTION;
Main.M51.bHardwareEnable      := TRUE;
Main.M51.bPowerSelf           := TRUE;
fbMotion3(stMotionStage:=Main.M51);

// Motor 4 RETICLE VERT Y (SP1L0-KMONO-MMS-04)
//Main.M52.bLimitForwardEnable  := bM4CWLimit;    //(+Y)
//Main.M52.bLimitBackwardEnable := bM4CCWLimit;    //(-Y)
Main.M52.nEnableMode          := Enum_StageEnableMode.ALWAYS;
Main.M52.bHardwareEnable      := TRUE;
Main.M52.bPowerSelf           := TRUE;
fbMotion4(stMotionStage:=Main.M52);
//fbFFO4(stMotionStage := Main.M52,
//       fbFFHWO := GVL.fbFastFaultOutput1);
// Andy says: trip reticle if not OUT
// OUT is 1.55843, in is high limit switch
// NOTE: we don't have an encoder or an LVDT on this axis! We will use the out switch
bRetOut := NOT Main.M52.bLimitForwardEnable;
fbRetFFO(
    i_xOk := bRetOut,
    i_xAutoReset := TRUE,
    i_DevName := Main.M52.sName,
    i_Desc := 'Reticle not OUT (y>0)',
    io_fbFFHWO := GVL.fbFastFaultOutput1);

// Motor 5 DIODE HORIZ X (SP1L0-KMONO-MMS-05)
//Main.M53.bLimitForwardEnable  := bM5CCWLimit;    //(+X)
//Main.M53.bLimitBackwardEnable := bM5CWLimit;    //(-X)
Main.M53.nEnableMode          := Enum_StageEnableMode.DURING_MOTION;
Main.M53.bHardwareEnable      := TRUE;
Main.M53.bPowerSelf           := TRUE;
fbMotion5(stMotionStage:=Main.M53);

// Motor 6 DIODE VERT Y (SP1L0-KMONO-MMS-06)
//Main.M54.bLimitForwardEnable  := bM6CWLimit;    //(+Y)
//Main.M54.bLimitBackwardEnable := bM6CCWLimit;    //(-Y)
Main.M54.nEnableMode          := Enum_StageEnableMode.ALWAYS;
Main.M54.bHardwareEnable      := TRUE;
Main.M54.bPowerSelf           := TRUE;
fbMotion6(stMotionStage:=Main.M54);
//fbFFO6(stMotionStage := Main.M54,
//       fbFFHWO := GVL.fbFastFaultOutput1);
// Andy says trip if NOT IN or NOT OUT
// Andy says trip if IN AND NOT (7.7 to 8.9 keV)
// IN is 0, OUT is 98.5
bDiodeOut := Main.M54.stAxisStatus.fActPosition > 96.5;
bDiodeIn := Main.M54.stAxisStatus.fActPosition < 2;
fbDiodeFFOAtPos(
    i_xOk := bDiodeOut XOR bDiodeIn,
    i_xAutoReset := TRUE,
    i_DevName := Main.M54.sName,
    i_Desc := 'Diode between states.',
    io_fbFFHWO := GVL.fbFastFaultOutput1);
fbDiodeFFOEnergy(
    i_xOk := bEnergyOk OR NOT bDiodeIn,
    i_xReset := bDiodeOut OR (bDiodeIn AND bEnergyOk),
    i_xAutoReset := TRUE,
    i_DevName := Main.M54.sName,
    //i_Desc := 'Unsafe eV Range',
    i_Desc := 'Override if 7.7-8.9keV',
    io_fbFFHWO := GVL.fbFastFaultOutput1);

END_PROGRAM

// ---- Temp/FB_BasicAxisFFO.TcPOU
FUNCTION_BLOCK FB_BasicAxisFFO
(*
    Placeholder FFO logic for no beam allowed, pre-comissioning

    Fast fault is applied if the axis is moving.
*)
VAR_IN_OUT
    Axis: AXIS_REF;
    fbFFHWO: FB_HardwareFFOutput;
END_VAR
VAR_INPUT
    sName: STRING;
END_VAR
VAR_OUTPUT
    bIsNotMoving: BOOL;
END_VAR
VAR
    fbFF: FB_FastFault := (i_Desc := 'Device is moving',
                           i_TypeCode := 16#2100,
                           i_xAutoReset := TRUE);
END_VAR

bIsNotMoving := NOT Axis.Status.Moving;
fbFF(i_DevName := sName,
     i_xOK := bIsNotMoving,
     io_fbFFHWO := fbFFHWO);

END_FUNCTION_BLOCK

// ---- Temp/FB_BasicMotionStageAltFFO.TcPOU
FUNCTION_BLOCK FB_BasicMotionStageAltFFO
(*
    Alternative to FB_BasicMotionStageFFO for an arbitrary out condition

    Sometimes the out limits is not what we want to use for proto-mps
*)
VAR_IN_OUT
    stMotionStage: DUT_MotionStage;
    fbFFHWO: FB_HardwareFFOutput;
END_VAR
VAR_INPUT
    sName: STRING;
    bFFOk: BOOL;
END_VAR
VAR_OUTPUT
    bIsOut: BOOL;
    bIsNotMoving: BOOL;
END_VAR
VAR
    fbBasicAxisFFO: FB_BasicAxisFFO := (sName := sName);
    fbFF: FB_FastFault := (i_Desc := 'Device is not out',
                           i_TypeCode := 16#2200,
                           i_xAutoReset := TRUE);
END_VAR

fbBasicAxisFFO(Axis := stMotionStage.Axis,
               fbFFHWO := fbFFHWO,
               sName := sName,
               bIsNotMoving => bIsNotMoving);

fbFF(i_DevName := sName,
     i_xOK := bFFOk,
     io_fbFFHWO := fbFFHWO);

END_FUNCTION_BLOCK

// ---- Temp/FB_BasicMotionStageFFO.TcPOU
FUNCTION_BLOCK FB_BasicMotionStageFFO
(*
    Placeholder FFO logic for no beam allowed, pre-comissioning

    Fast fault is applied if the motor is moving or is not at the out switch.
*)
VAR_IN_OUT
    stMotionStage: DUT_MotionStage;
    fbFFHWO: FB_HardwareFFOutput;
END_VAR
VAR_INPUT
    sName: STRING;
    bForwardIsOut: BOOL := TRUE;
END_VAR
VAR_OUTPUT
    bIsOut: BOOL;
    bIsNotMoving: BOOL;
END_VAR
VAR
    fbBasicAxisFFO: FB_BasicAxisFFO := (sName := sName);
    fbFF: FB_FastFault := (i_Desc := 'Device is not out',
                           i_TypeCode := 16#2200,
                           i_xAutoReset := TRUE);
END_VAR

fbBasicAxisFFO(Axis := stMotionStage.Axis,
               fbFFHWO := fbFFHWO,
               sName := sName,
               bIsNotMoving => bIsNotMoving);

IF bForwardIsOut THEN
    bIsOut := NOT stMotionStage.bLimitForwardEnable;
ELSE
    bIsOut := NOT stMotionStage.bLimitBackwardEnable;
END_IF

fbFF(i_DevName := sName,
     i_xOK := bIsOut,
     io_fbFFHWO := fbFFHWO);

END_FUNCTION_BLOCK

// ---- Temp/FB_SimMotor.TcPOU
FUNCTION_BLOCK FB_SimMotor
VAR_IN_OUT
    stMotionStage: DUT_MotionStage;
END_VAR
VAR
    fbMotionStage: FB_MotionStage;
END_VAR

stMotionStage.bLimitBackwardEnable := TRUE;
stMotionStage.bLimitForwardEnable := TRUE;
stMotionStage.bHardwareEnable := TRUE;
stMotionStage.bPowerSelf := TRUE;
stMotionStage.nEnableMode := ENUM_StageEnableMode.ALWAYS;
fbMotionStage(stMotionStage := stMotionStage);

END_FUNCTION_BLOCK
